Fanuc KAREL source: ko00061.KL

-- PROVISIONAL review KL for V770-1; original PC SHA256 da00c30b9340afd0bf507a3365704ff2f743e68ea2b203dadd8b1e0c3fe6bc85
-- Incomplete behavior may be omitted. Consult companion uncertainty JSON. Do not deploy.
PROGRAM KO00061
%NOLOCKGROUP
BEGIN
  -- UNRESOLVED_PC offsets 5-12; opcodes 9D,23
  -- UNRESOLVED_PC offsets 17-69; opcodes 27,27,49,7E,AD,27,49,7E,AD,22,31,7E,4A
  -- UNRESOLVED_PC offsets 74-78; opcodes 7F
END KO00061
